// Mitsubishi GX Works2 project: 20150604   PLC: Q03UDV

PROGRAM 1
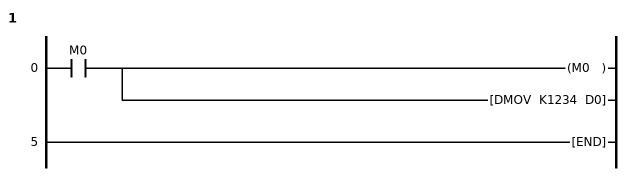
0     LD      M0
      OUT     M0
      DMOV    K1234 D0
5     END
END_PROGRAM

PROGRAM 2
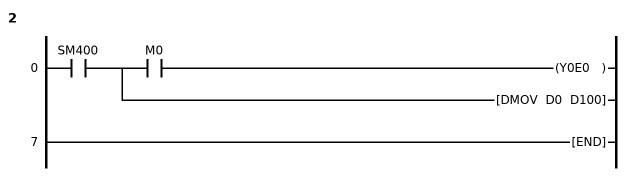
0     LD      SM400
      MPS
      AND     M0
      OUT     Y0E0
      MPP
      DMOV    D0 D100
7     END
END_PROGRAM
